FUNCTION_BLOCK Sensor_NClose IMPLEMENTS I_Sensor
VAR
	bInput AT %I* : BOOL;
END_VAR

PROPERTY isActive : BOOL
GET
isActive:= not bInput;
END_GET
END_PROPERTY

PROPERTY notActive : BOOL
GET
isActive := bInput;
END_GET
END_PROPERTY

END_FUNCTION_BLOCK

(* stored: Version 1.1.0.1, ProductVersion 3.1.4024.12
   POU Sensor_NClose: Id {f6f1ca14-2fe4-4d15-9932-61636ed7cf4a}, SpecialFunc None
   Property isActive: Id {fa14f7d1-9931-4481-aef8-1bfb71f540bd}
   Get Get: Id {b8924d53-115a-44c0-9e78-c8cb723bf907}
   Property notActive: Id {a0d9e939-ff52-4ece-8594-ba4894b9c6fe}
   Get Get: Id {5367e314-78d1-42be-b8e8-9cdb4c9b8399} *)
